// Mitsubishi GX Works2 project: EXE2_Group7   PLC: FX3G

// global labels: Global1
VAR_GLOBAL
  startLisha AT X001 : BOOL;
  StartkneadingDough AT X002 : BOOL;
  qualityCheck AT X003 : BOOL;
  flourQuantity AT D1100 : REAL;
  yeastQuantity AT D1102 : REAL;
  waterQuantity AT D1104 : REAL;
  oilQuantity AT D1106 : REAL;
  spicesQuantity AT D1108 : REAL;
  timerY5 AT TC0 : BOOL;
  helperY5 AT TS0 : BOOL;
  helperY6 AT TS1 : BOOL;
  timerY6 AT TC1 : BOOL;
  BreadShelfCount AT D1110 : INT;
  timerY2 AT TC2 : BOOL;
  helperY2 AT TS2 : BOOL;
  timerY3 AT TC3 : BOOL;
  helperY3 AT TS3 : BOOL;
  timerY2Y3 AT TS4 : BOOL;
  helperY2Y3 AT TC4 : BOOL;
  timerY4 AT TC5 : BOOL;
  helperY4 AT TS5 : BOOL;
  stopDay AT X007 : BOOL;
  startDay AT X010 : BOOL;
  hatpahaStart AT X011 : BOOL;
  timerY10Stop AT TC6 : BOOL;
  helperY10Stop AT TS6 : BOOL;
  hatpahaLamp1 AT Y002 : BOOL;
  hatpahaLamp2 AT Y003 : BOOL;
  BakingLamp AT Y004 : BOOL;
  KneadingDoughLamp AT Y005 : BOOL;
  QualityCheckLamp AT Y006 : BOOL;
  dayLamp AT Y010 : BOOL;
  countX11 AT CS0 : BOOL;
  counterX11 AT CC0 : BOOL;
  helperY10blink AT TC7 : BOOL;
  timerY10 AT TS7 : BOOL;
  timeY10Blink1 AT TC8 : BOOL;
  helperY10Blink1 AT TS8 : BOOL;
  timerY10Blink2 AT TC9 : BOOL;
  helperY10Blink2 AT TS9 : BOOL;
  LishaLamp AT Y001 : BOOL;
  Bowl AT D1112 : REAL;
  BakingPan AT D1114 : REAL;
  mixer AT D1116 : REAL;
  hatpahaPan AT D1118 : REAL;
  counterM13 AT CC1 : BOOL;
  countM13 AT CS1 : BOOL;
  doneProcess AT M1 : BOOL;
  checkQuantity AT M2 : BOOL;
  helperOKanalog AT M3 : BOOL;
  helperCheckRatioQuantity AT M4 : BOOL;
  helperKneadingDough AT M5 : BOOL;
  helperBaking AT M6 : BOOL;
  HelperDoneProcess AT M7 : BOOL;
  healperQualityCheck AT M8 : BOOL;
  helperLampY1 AT M9 : BOOL;
  helperTimerY6 AT M10 : BOOL;
  HelperBreadCount AT M11 : BOOL;
  HelperHatpaha AT M12 : BOOL;
  helperCantProduce AT M13 : BOOL;
  helperStartBaking AT M14 : BOOL;
  helperNotOKanalog AT M15 : BOOL;
  ratioHappend AT M16 : BOOL;
  helperAddBreadToShelf AT M17 : BOOL;
  helperProduce AT M18 : BOOL;
  productTaken AT M19 : BOOL;
  helperThrowBread AT M20 : BOOL;
  cantProduce AT M23 : BOOL;
  canProduce AT M24 : BOOL;
  ratioNotHappend AT M25 : BOOL;
  HelperDayON AT M29 : BOOL;
  finishDay AT M30 : BOOL;
  helperFinishDay AT M31 : BOOL;
  HelperEndDayBlinkLamp AT M32 : BOOL;
  HelperWorkDay AT M36 : BOOL;
  fakeLamp AT M40 : BOOL;
END_VAR
VAR_GLOBAL CONSTANT
  constant1 : INT := 1;
  constant2 : INT := 2;
  constant3 : INT := 3;
  constant4 : INT := 4;
  constant5 : INT := 5;
  constant30 : INT := 30;
  constant40 : INT := 40;
  constant50 : INT := 50;
  constant150 : INT := 150;
  constant1Analog : INT := 400;
  constant5Analog : INT := 2000;
  constantF0 : REAL;
  constantF0_1 : REAL := 0.1;
  constantF0_2 : REAL := 0.2;
  constantF0_3 : REAL := 0.3;
  constantF0_5 : REAL := 0.5;
  constantF1 : REAL := 1;
  constantF10 : REAL := 10;
  constantF20 : REAL := 20;
  constantF30 : REAL := 30;
  constantF50 : REAL := 50;
  constantF100 : REAL := 100;
  constantAllProductsF210 : REAL := 210;
  constantF500 : REAL := 500;
END_VAR
VAR_GLOBAL
  InputFlourQuantity AT D1120 : REAL;
  inputYeastQuantity AT D1122 : REAL;
  inputWaterQuantity AT D1124 : REAL;
  inputOilQuantity AT D1126 : REAL;
  inputSpicesQuantity AT D1128 : REAL;
  analog_input_2 AT D8281 : INT;
END_VAR

// task Task_01 (event TRUE, interval 0, priority 31): POU_01

PROGRAM POU_01
(* structured ladder/FBD written out as ST: instructions are called as NAME(EN, inputs, outputs); _pN, _eN, _tN stand for wires *)
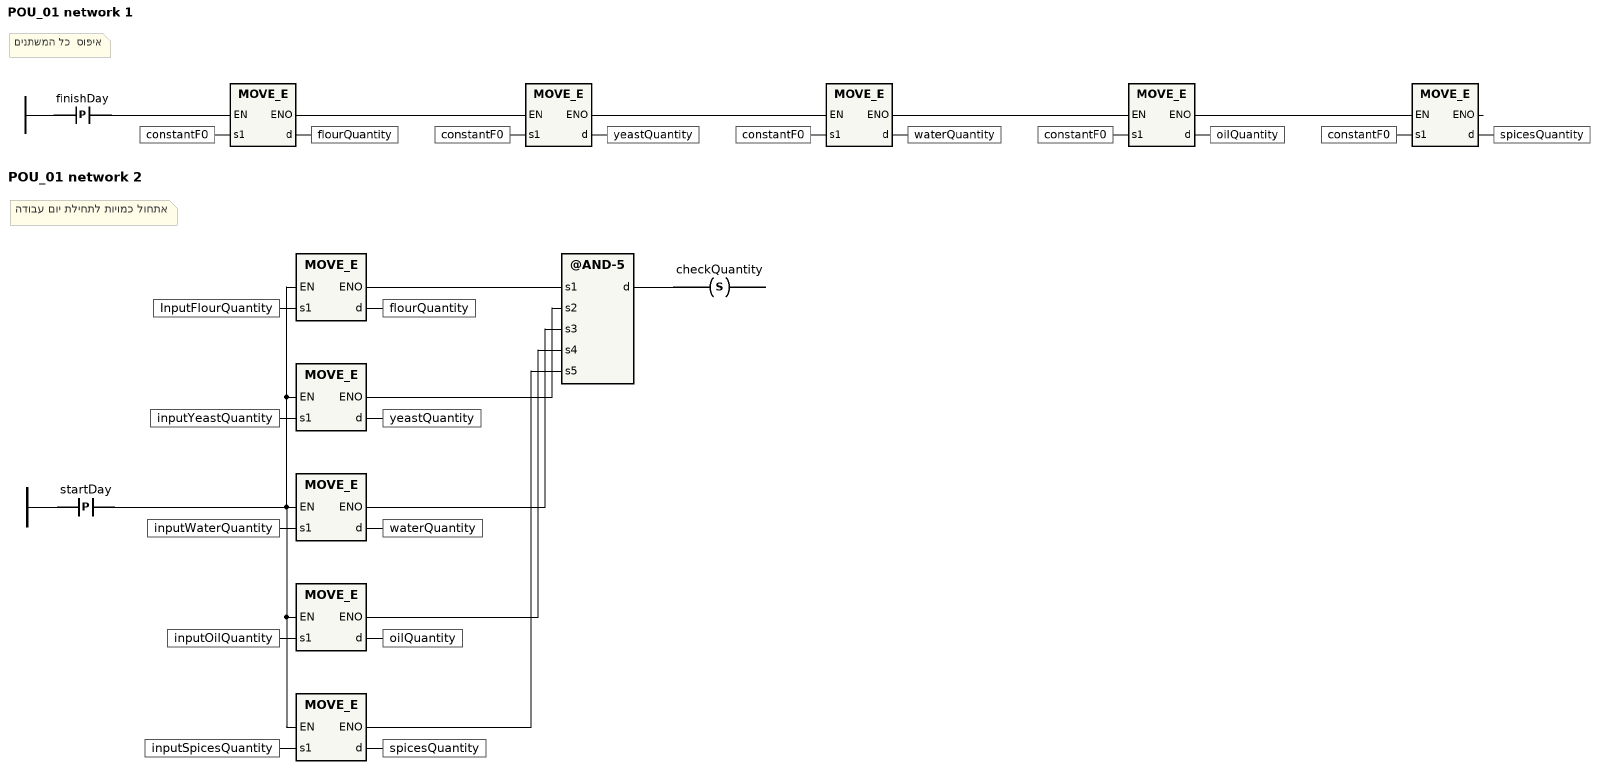
(* network 1 *)
(* איפוס  כל המשתנים *)
_e1 := MOVE_E(LDP(TRUE, finishDay), constantF0, flourQuantity);
_e2 := MOVE_E(_e1, constantF0, yeastQuantity);
_e3 := MOVE_E(_e2, constantF0, waterQuantity);
_e4 := MOVE_E(_e3, constantF0, oilQuantity);
MOVE_E(_e4, constantF0, spicesQuantity);
(* network 2 *)
(* אתחול כמויות לתחילת יום עבודה *)
_p1 := LDP(TRUE, startDay);
_e2 := MOVE_E(_p1, InputFlourQuantity, flourQuantity);
_e3 := MOVE_E(_p1, inputYeastQuantity, yeastQuantity);
_e4 := MOVE_E(_p1, inputWaterQuantity, waterQuantity);
_e5 := MOVE_E(_p1, inputOilQuantity, oilQuantity);
_e6 := MOVE_E(_p1, inputSpicesQuantity, spicesQuantity);
SET(@AND-5(_e2, _e3, _e4, _e5, _e6), checkQuantity);
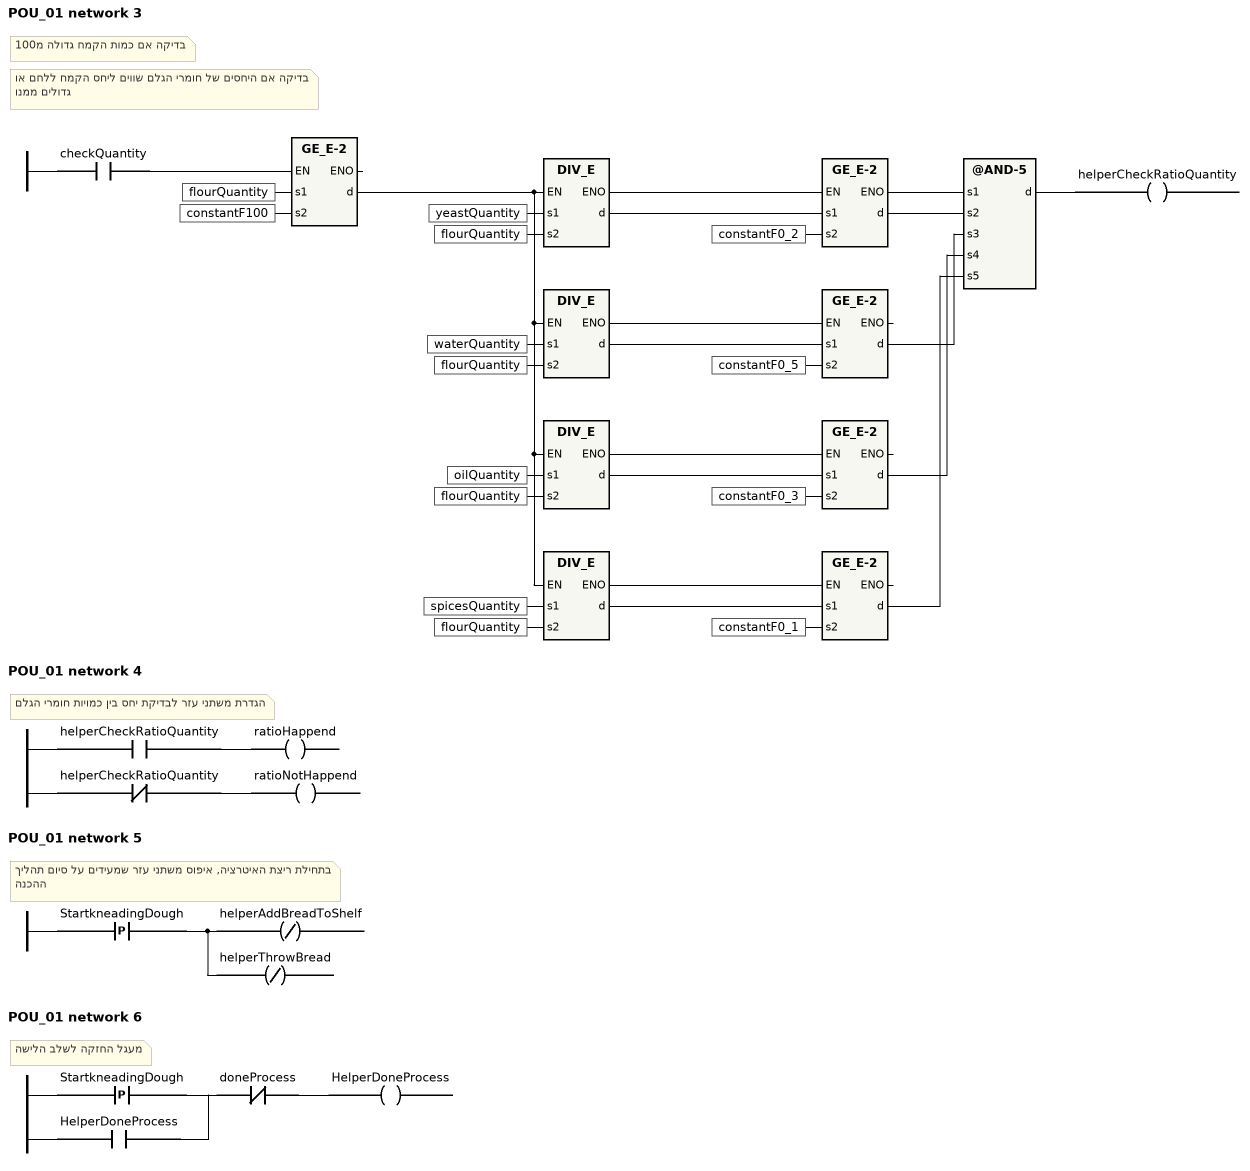
(* network 3 *)
(* בדיקה אם כמות הקמח גדולה מ100 *)
(* בדיקה אם היחסים של חומרי הגלם שווים ליחס הקמח ללחם או גדולים ממנו *)
GE_E(checkQuantity, flourQuantity, constantF100, _t1);
_e3 := DIV_E(_t1, yeastQuantity, flourQuantity, _t2);
_e5 := GE_E(_e3, _t2, constantF0_2, _t4);
_e7 := DIV_E(_t1, waterQuantity, flourQuantity, _t6);
GE_E(_e7, _t6, constantF0_5, _t8);
_e10 := DIV_E(_t1, oilQuantity, flourQuantity, _t9);
GE_E(_e10, _t9, constantF0_3, _t11);
_e13 := DIV_E(_t1, spicesQuantity, flourQuantity, _t12);
GE_E(_e13, _t12, constantF0_1, _t14);
helperCheckRatioQuantity := @AND-5(_e5, _t4, _t8, _t11, _t14);
(* network 4 *)
(* הגדרת משתני עזר לבדיקת יחס בין כמויות חומרי הגלם *)
ratioHappend := helperCheckRatioQuantity;
ratioNotHappend := NOT helperCheckRatioQuantity;
(* network 5 *)
(* בתחילת ריצת האיטרציה, איפוס משתני עזר שמעידים על סיום תהליך ההכנה *)
_p1 := LDP(TRUE, StartkneadingDough);
helperAddBreadToShelf := NOT _p1;
helperThrowBread := NOT _p1;
(* network 6 *)
(* מעגל החזקה לשלב הלישה *)
HelperDoneProcess := (LDP(TRUE, StartkneadingDough) OR HelperDoneProcess) AND NOT doneProcess;
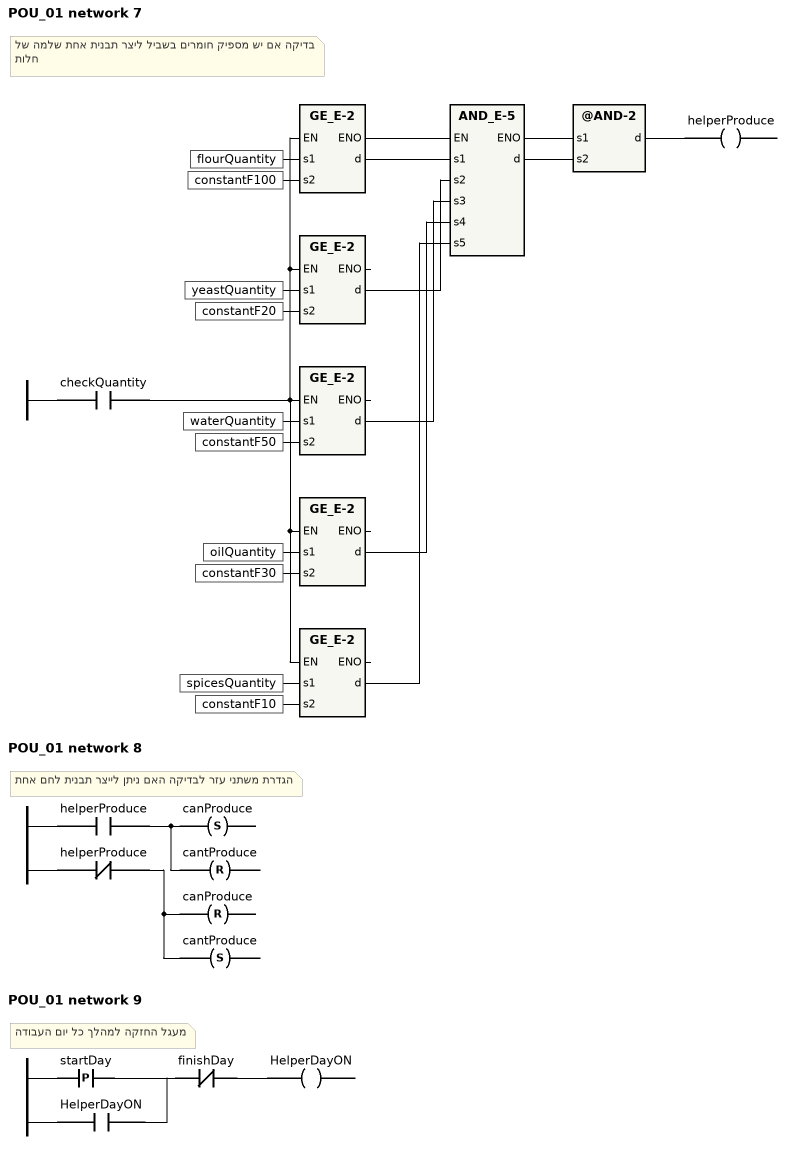
(* network 7 *)
(* בדיקה אם יש מספיק חומרים בשביל ליצר תבנית אחת שלמה של חלות *)
_e2 := GE_E(checkQuantity, flourQuantity, constantF100, _t1);
GE_E(checkQuantity, yeastQuantity, constantF20, _t3);
GE_E(checkQuantity, waterQuantity, constantF50, _t4);
GE_E(checkQuantity, oilQuantity, constantF30, _t5);
GE_E(checkQuantity, spicesQuantity, constantF10, _t6);
_e8 := AND_E(_e2, _t1, _t3, _t4, _t5, _t6, _t7);
helperProduce := @AND-2(_e8, _t7);
(* network 8 *)
(* הגדרת משתני עזר לבדיקה האם ניתן לייצר תבנית לחם אחת *)
SET(helperProduce, canProduce);
RST(helperProduce, cantProduce);
_p1 := NOT helperProduce;
RST(_p1, canProduce);
SET(_p1, cantProduce);
(* network 9 *)
(* מעגל החזקה למהלך כל יום העבודה *)
HelperDayON := (LDP(TRUE, startDay) OR HelperDayON) AND NOT finishDay;
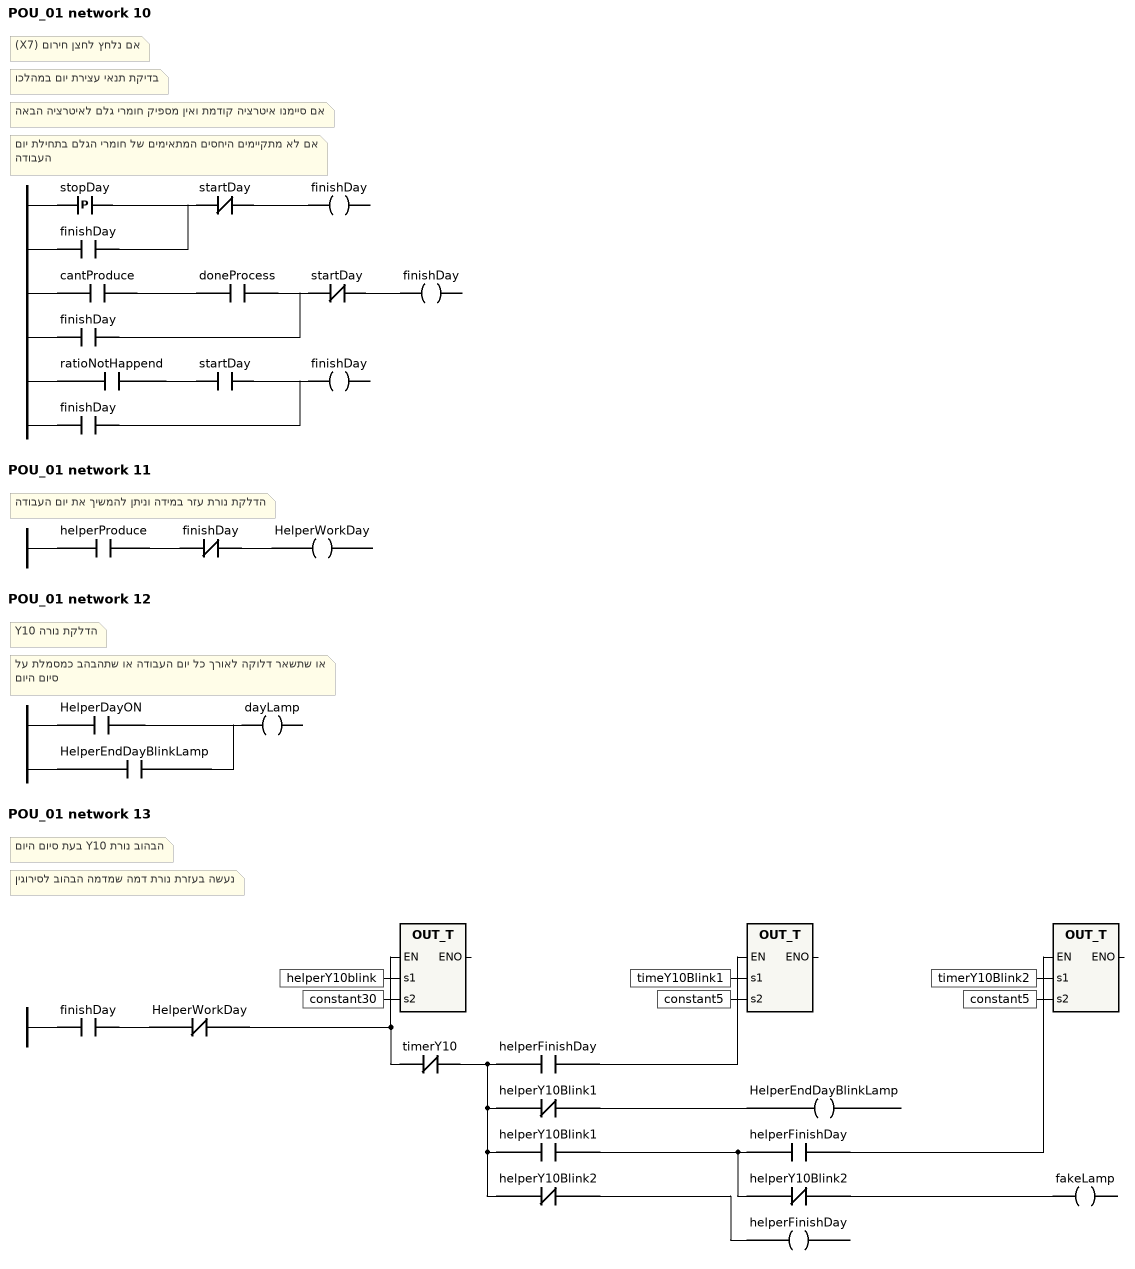
(* network 10 *)
(* אם נלחץ לחצן חירום (X7) *)
(* בדיקת תנאי עצירת יום במהלכו *)
(* אם סיימנו איטרציה קודמת ואין מספיק חומרי גלם לאיטרציה הבאה *)
(* אם לא מתקיימים היחסים המתאימים של חומרי הגלם בתחילת יום העבודה *)
finishDay := (LDP(TRUE, stopDay) OR finishDay) AND NOT startDay;
finishDay := ((cantProduce AND doneProcess) OR finishDay) AND NOT startDay;
finishDay := (ratioNotHappend AND startDay) OR finishDay;
(* network 11 *)
(* הדלקת נורת עזר במידה וניתן להמשיך את יום העבודה *)
HelperWorkDay := helperProduce AND NOT finishDay;
(* network 12 *)
(* הדלקת נורה Y10 *)
(* או שתשאר דלוקה לאורך כל יום העבודה או שתהבהב כמסמלת על סיום היום *)
dayLamp := HelperDayON OR HelperEndDayBlinkLamp;
(* network 13 *)
(* הבהוב נורת Y10 בעת סיום היום *)
(* נעשה בעזרת נורת דמה שמדמה הבהוב לסירוגין *)
_p1 := finishDay AND NOT HelperWorkDay;
OUT_T(_p1, helperY10blink, constant30);
_p2 := _p1 AND NOT timerY10;
OUT_T(_p2 AND helperFinishDay, timeY10Blink1, constant5);
HelperEndDayBlinkLamp := _p2 AND NOT helperY10Blink1;
_p3 := _p2 AND helperY10Blink1;
OUT_T(_p3 AND helperFinishDay, timerY10Blink2, constant5);
fakeLamp := _p3 AND NOT helperY10Blink2;
helperFinishDay := _p2 AND NOT helperY10Blink2;
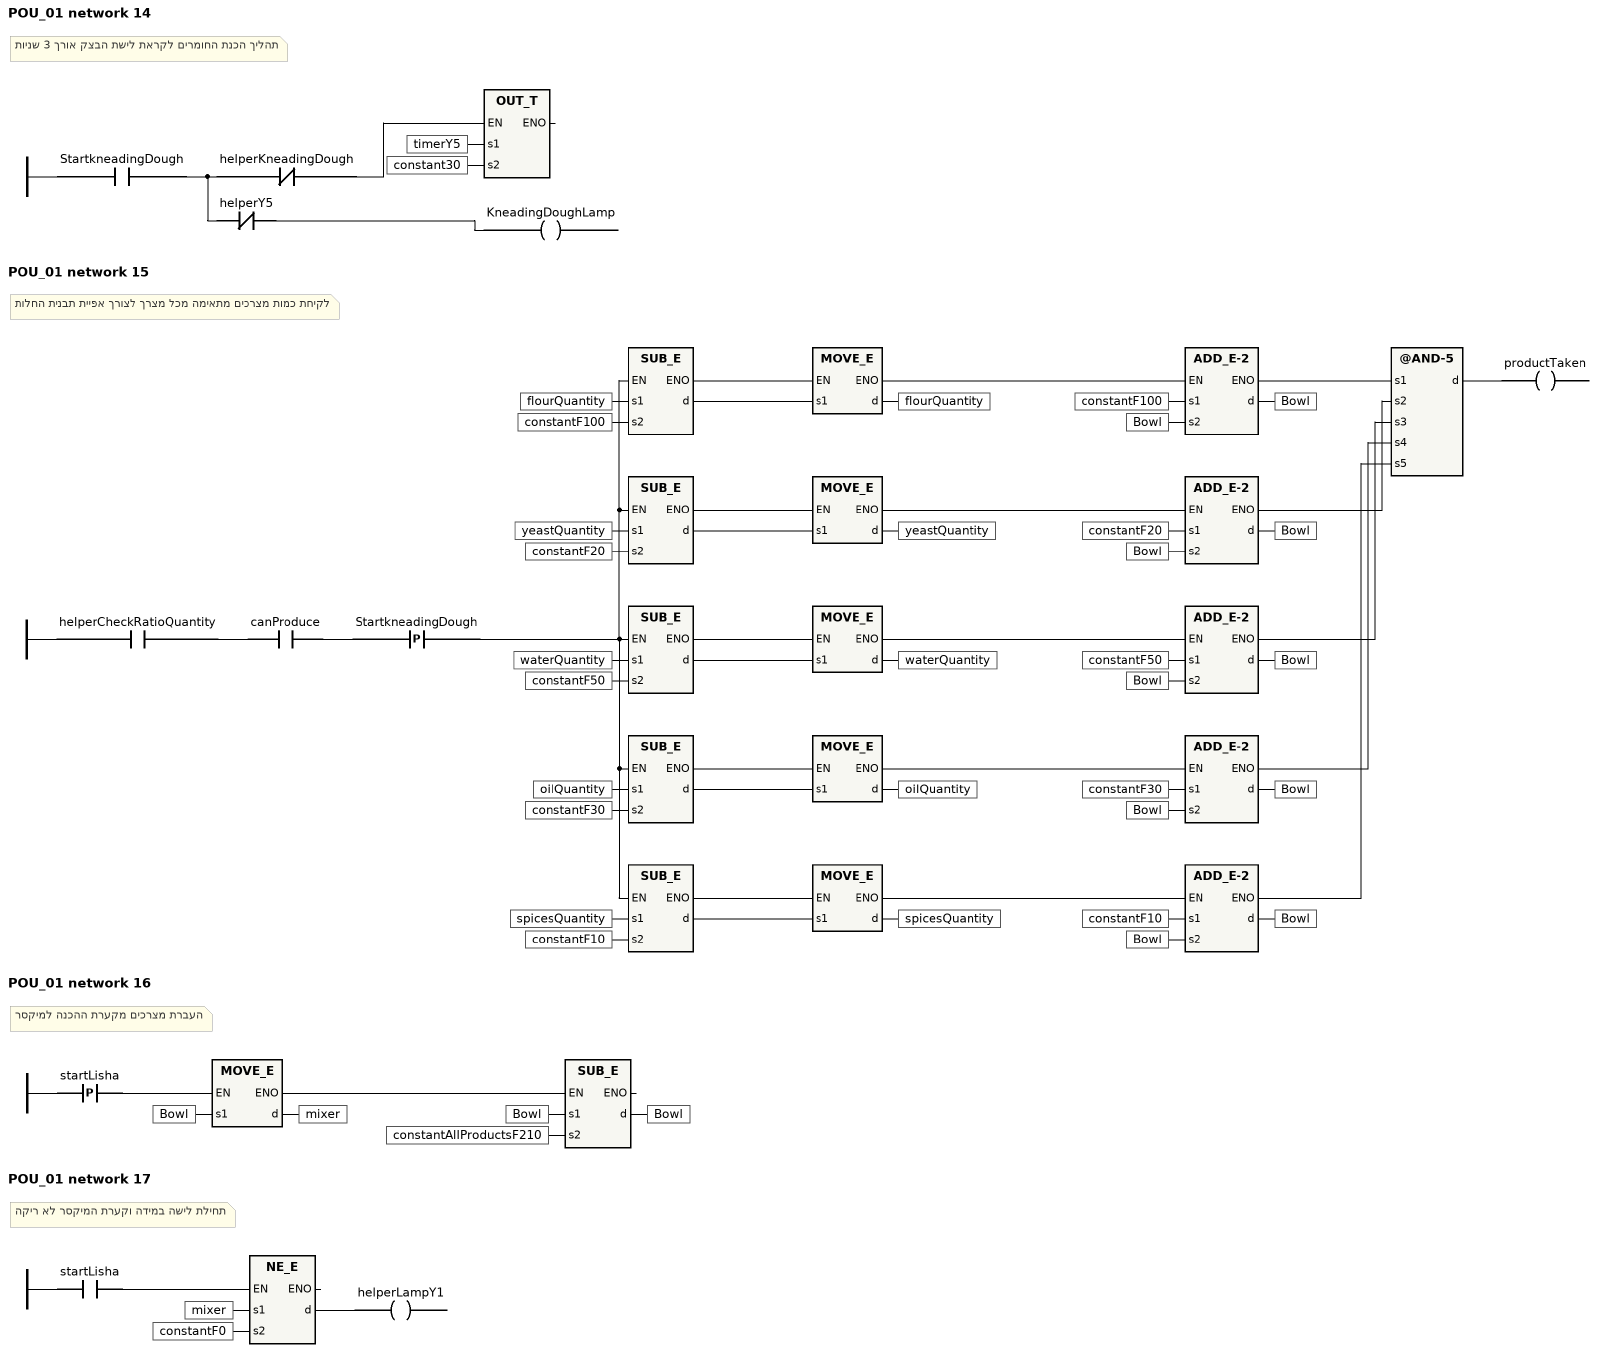
(* network 14 *)
(* תהליך הכנת החומרים לקראת לישת הבצק אורך 3 שניות *)
OUT_T(StartkneadingDough AND NOT helperKneadingDough, timerY5, constant30);
KneadingDoughLamp := StartkneadingDough AND NOT helperY5;
(* network 15 *)
(* לקיחת כמות מצרכים מתאימה מכל מצרך לצורך אפיית תבנית החלות *)
_p1 := helperCheckRatioQuantity AND canProduce AND LDP(TRUE, StartkneadingDough);
_e3 := SUB_E(_p1, flourQuantity, constantF100, _t2);
_e4 := MOVE_E(_e3, _t2, flourQuantity);
_e5 := ADD_E(_e4, constantF100, Bowl, Bowl);
_e7 := SUB_E(_p1, yeastQuantity, constantF20, _t6);
_e8 := MOVE_E(_e7, _t6, yeastQuantity);
_e9 := ADD_E(_e8, constantF20, Bowl, Bowl);
_e11 := SUB_E(_p1, waterQuantity, constantF50, _t10);
_e12 := MOVE_E(_e11, _t10, waterQuantity);
_e13 := ADD_E(_e12, constantF50, Bowl, Bowl);
_e15 := SUB_E(_p1, oilQuantity, constantF30, _t14);
_e16 := MOVE_E(_e15, _t14, oilQuantity);
_e17 := ADD_E(_e16, constantF30, Bowl, Bowl);
_e19 := SUB_E(_p1, spicesQuantity, constantF10, _t18);
_e20 := MOVE_E(_e19, _t18, spicesQuantity);
_e21 := ADD_E(_e20, constantF10, Bowl, Bowl);
productTaken := @AND-5(_e5, _e9, _e13, _e17, _e21);
(* network 16 *)
(* העברת מצרכים מקערת ההכנה למיקסר *)
_e1 := MOVE_E(LDP(TRUE, startLisha), Bowl, mixer);
SUB_E(_e1, Bowl, constantAllProductsF210, Bowl);
(* network 17 *)
(* תחילת לישה במידה וקערת המיקסר לא ריקה *)
NE_E(startLisha, mixer, constantF0, _t1);
helperLampY1 := _t1;
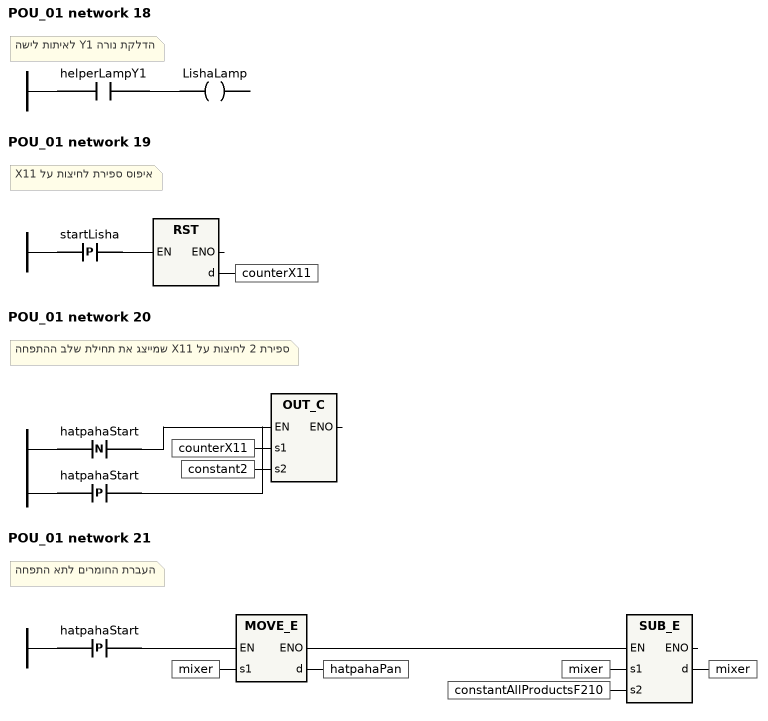
(* network 18 *)
(* הדלקת נורה Y1 לאיתות לישה *)
LishaLamp := helperLampY1;
(* network 19 *)
(* איפוס ספירת לחיצות על X11 *)
RST(LDP(TRUE, startLisha), counterX11);
(* network 20 *)
(* ספירת 2 לחיצות על X11 שמייצג את תחילת שלב ההתפחה *)
OUT_C(LDF(TRUE, hatpahaStart) OR LDP(TRUE, hatpahaStart), counterX11, constant2);
(* network 21 *)
(* העברת החומרים לתא התפחה *)
_e1 := MOVE_E(LDP(TRUE, hatpahaStart), mixer, hatpahaPan);
SUB_E(_e1, mixer, constantAllProductsF210, mixer);
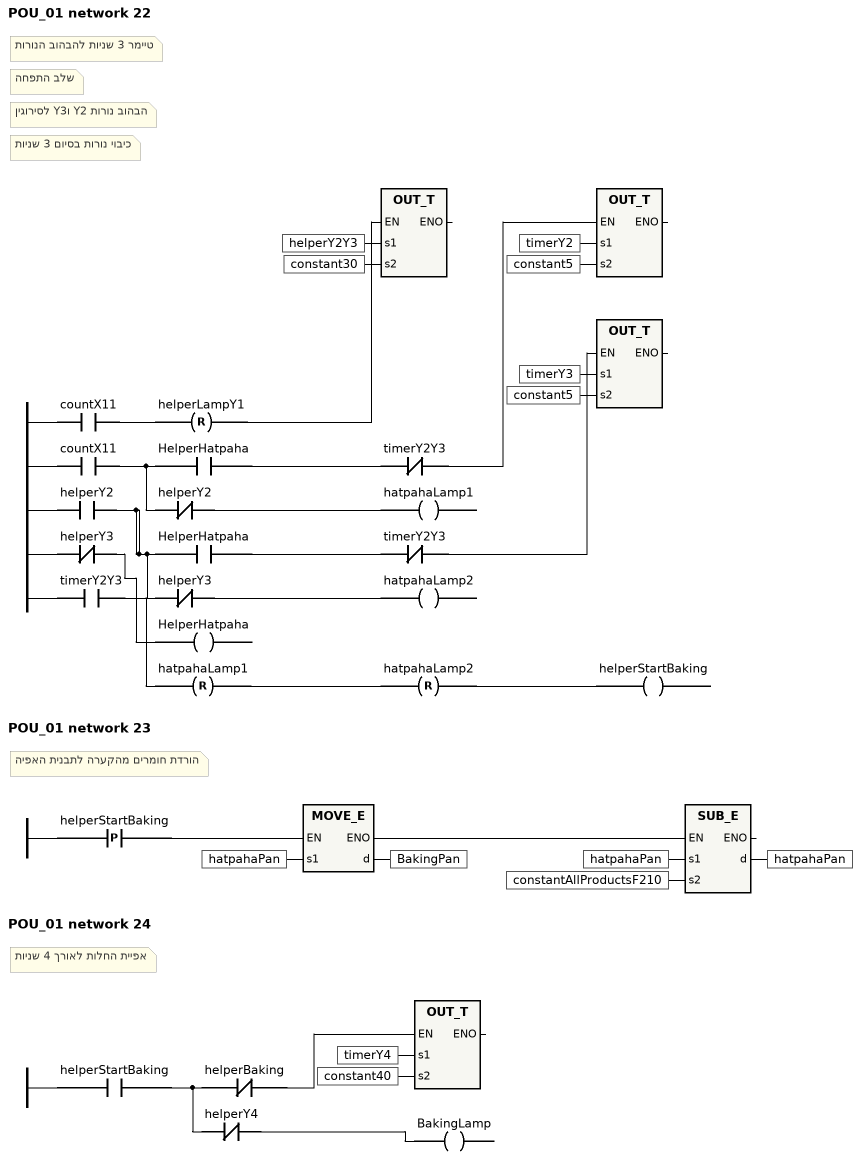
(* network 22 *)
(* טיימר 3 שניות להבהוב הנורות *)
(* שלב התפחה *)
(* הבהוב נורות Y2 וY3 לסירוגין *)
(* כיבוי נורות בסיום 3 שניות *)
RST(countX11, helperLampY1);
OUT_T(countX11, helperY2Y3, constant30);
OUT_T(countX11 AND HelperHatpaha AND NOT timerY2Y3, timerY2, constant5);
hatpahaLamp1 := countX11 AND NOT helperY2;
OUT_T(helperY2 AND HelperHatpaha AND NOT timerY2Y3, timerY3, constant5);
hatpahaLamp2 := helperY2 AND NOT helperY3;
HelperHatpaha := NOT helperY3;
RST(timerY2Y3, hatpahaLamp1);
RST(timerY2Y3, hatpahaLamp2);
helperStartBaking := timerY2Y3;
(* network 23 *)
(* הורדת חומרים מהקערה לתבנית האפיה *)
_e1 := MOVE_E(LDP(TRUE, helperStartBaking), hatpahaPan, BakingPan);
SUB_E(_e1, hatpahaPan, constantAllProductsF210, hatpahaPan);
(* network 24 *)
(* אפיית החלות לאורך 4 שניות *)
OUT_T(helperStartBaking AND NOT helperBaking, timerY4, constant40);
BakingLamp := helperStartBaking AND NOT helperY4;
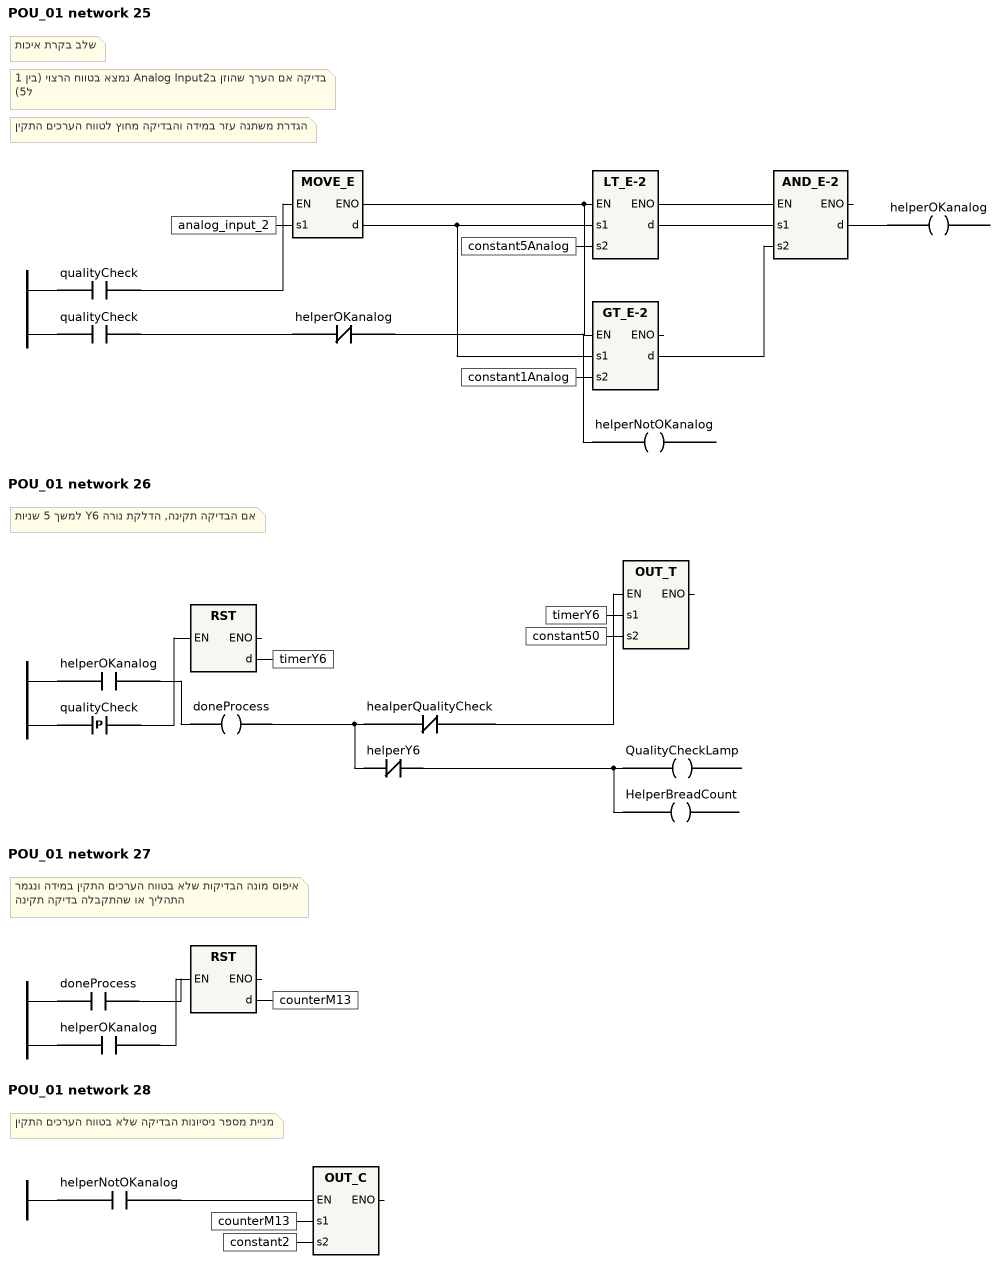
(* network 25 *)
(* שלב בקרת איכות *)
(* בדיקה אם הערך שהוזן בAnalog Input2 נמצא בטווח הרצוי (בין 1 ל5) *)
(* הגדרת משתנה עזר במידה והבדיקה מחוץ לטווח הערכים התקין *)
_e2 := MOVE_E(qualityCheck, analog_input_2, _t1);
_e4 := LT_E(_e2, _t1, constant5Analog, _t3);
GT_E(_e2, _t1, constant1Analog, _t5);
AND_E(_e4, _t3, _t5, _t6);
helperOKanalog := _t6;
helperNotOKanalog := qualityCheck AND NOT helperOKanalog;
(* network 26 *)
(* אם הבדיקה תקינה, הדלקת נורה Y6 למשך 5 שניות *)
doneProcess := helperOKanalog;
OUT_T(helperOKanalog AND NOT healperQualityCheck, timerY6, constant50);
_p1 := helperOKanalog AND NOT helperY6;
QualityCheckLamp := _p1;
HelperBreadCount := _p1;
RST(LDP(TRUE, qualityCheck), timerY6);
(* network 27 *)
(* איפוס מונה הבדיקות שלא בטווח הערכים התקין במידה ונגמר התהליך או שהתקבלה בדיקה תקינה *)
RST(doneProcess OR helperOKanalog, counterM13);
(* network 28 *)
(* מניית מספר ניסיונות הבדיקה שלא בטווח הערכים התקין *)
OUT_C(helperNotOKanalog, counterM13, constant2);
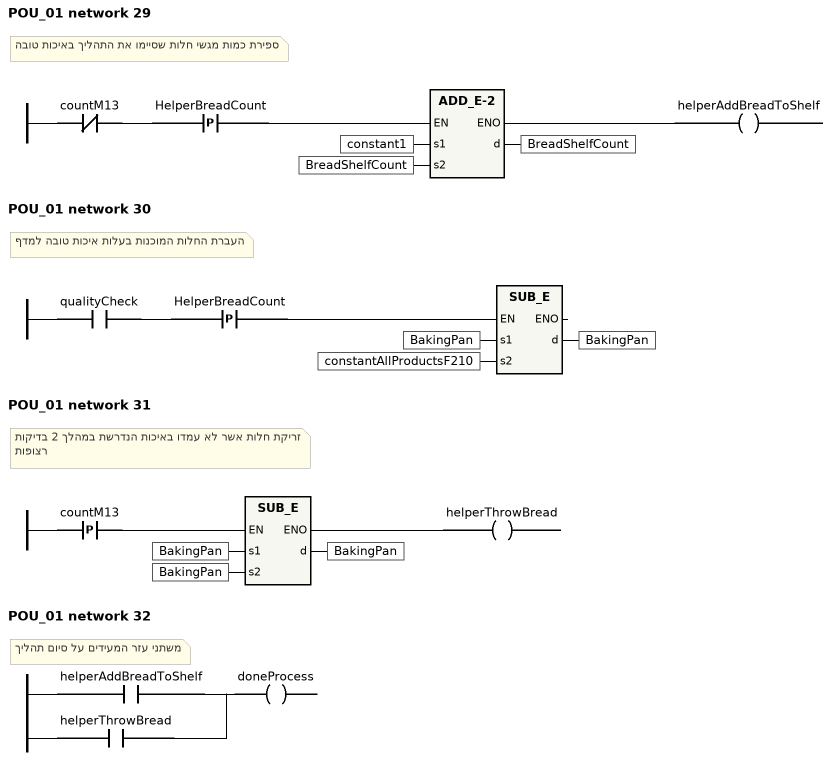
(* network 29 *)
(* ספירת כמות מגשי חלות שסיימו את התהליך באיכות טובה *)
_e1 := ADD_E(NOT countM13 AND LDP(TRUE, HelperBreadCount), constant1, BreadShelfCount, BreadShelfCount);
helperAddBreadToShelf := _e1;
(* network 30 *)
(* העברת החלות המוכנות בעלות איכות טובה למדף *)
SUB_E(qualityCheck AND LDP(TRUE, HelperBreadCount), BakingPan, constantAllProductsF210, BakingPan);
(* network 31 *)
(* זריקת חלות אשר לא עמדו באיכות הנדרשת במהלך 2 בדיקות רצופות *)
_e1 := SUB_E(LDP(TRUE, countM13), BakingPan, BakingPan, BakingPan);
helperThrowBread := _e1;
(* network 32 *)
(* משתני עזר המעידים על סיום תהליך *)
doneProcess := helperAddBreadToShelf OR helperThrowBread;
END_PROGRAM
